TYPE ST_AutoMode_ShippingLeftSideTransCV :
STRUCT
	Command : ST_CommandBasic;
	Status	: ST_StatusBasic;
	ShippingTransCVRequest_LeftSide : BOOL;		//C# to PLC
END_STRUCT
END_TYPE

(* stored: Version 1.1.0.1, ProductVersion 3.1.4024.13
   DUT ST_AutoMode_ShippingLeftSideTransCV: Id {cb837d1e-ab78-47a3-a1a9-a3e55298099e} *)
